TYPE ST_AI :
STRUCT
		Value		  AT %I*	: INT	;
		Description 			: STRING	;

END_STRUCT
END_TYPE

(* stored: Version 1.1.0.1, ProductVersion 3.1.4022.11
   DUT ST_AI: Id {1bada066-188a-4fe5-a5b4-2cdc70da015f} *)
